// TIA Portal V20 export
FUNCTION_BLOCK "Sequence_1_UnWinder"   // FB118, LAD
TITLE = Sequence
// Sequence template programmend in ladder logic
// stored: IsIECCheckEnabled true, MemoryReserve 100, Namespace Unit1.Em1, SetENOAutomatically true
   VAR
      instSequenceLADControl { ExternalWritable := 'False'} : "LAF_ControlLadSequence";
      instSequenceLADStatus { ExternalWritable := 'False'} : "LAF_StatusLadSequence";
      statPulse { ExternalWritable := 'False'} : Array[0..999] of Bool;
      statTonTimer { ExternalWritable := 'False'} : Array[0..999] of TON_TIME;
   END_VAR
   VAR_TEMP
      tempCustomerAction : Bool;   // Placeholder for possible actions
      tempDo_nothing_and_wait_for_init : Bool;   // Placeholder for doing nothing
      tempSafeStateCondition : Bool;   // Temp Condition for the equipment module to be in a safe state
   END_VAR
   VAR CONSTANT
      STEP_IDLE : DInt := 1;   // Idle Step
      JOB_1_STEP_01 : DInt := 101;
      JOB_1_STEP_11 : DInt := 111;
      JOB_1_STEP_21 : DInt := 121;
      JOB_1_STEP_31 : DInt := 131;
      JOB_1_STEP_41 : DInt := 141;
      JOB_1_STEP_51 : DInt := 151;
      JOB_1_STEP_61 : DInt := 161;
      JOB_1_STEP_71 : DInt := 171;
      JOB_1_STEP_81 : DInt := 181;
      JOB_1_STEP_91 : DInt := 191;
      JOB_2_STEP_01 : DInt := 201;
      JOB_2_STEP_11 : DInt := 211;
      JOB_2_STEP_21 : DInt := 221;
      JOB_2_STEP_31 : DInt := 231;
      JOB_2_STEP_41 : DInt := 241;
      JOB_2_STEP_51 : DInt := 251;
      JOB_2_STEP_61 : DInt := 261;
      JOB_2_STEP_71 : DInt := 271;
      JOB_2_STEP_81 : DInt := 281;
      JOB_2_STEP_91 : DInt := 291;
      JOB_3_STEP_01 : DInt := 301;
      JOB_3_STEP_11 : DInt := 311;
      JOB_3_STEP_21 : DInt := 321;
      JOB_3_STEP_31 : DInt := 331;
      JOB_3_STEP_41 : DInt := 341;
      JOB_3_STEP_51 : DInt := 351;
      JOB_3_STEP_61 : DInt := 361;
      JOB_3_STEP_71 : DInt := 371;
      JOB_3_STEP_81 : DInt := 381;
      JOB_3_STEP_91 : DInt := 391;
      JOB_4_STEP_01 : DInt := 401;
      JOB_4_STEP_11 : DInt := 411;
      JOB_4_STEP_21 : DInt := 421;
      JOB_4_STEP_31 : DInt := 431;
      JOB_4_STEP_41 : DInt := 441;
      JOB_4_STEP_51 : DInt := 451;
      JOB_4_STEP_61 : DInt := 461;
      JOB_4_STEP_71 : DInt := 471;
      JOB_4_STEP_81 : DInt := 481;
      JOB_4_STEP_91 : DInt := 491;
      STEP_IMMEDIATE_STOP : DInt := 901;   // Step executed when an immediate stop command is triggered for the sequence (i.e. when unit is in state aborting)
      SeqDelayTime : Time := T#100ms;
      SeqNoDelayTime : Time;
      SeqReWindingTime : Time := T#3s;
      TRUE : Bool := TRUE;
      FALSE : Bool := FALSE;
   END_VAR
   VAR_TEMP   // added for the SCL form of the ladder/FBD networks
      _w1 : Bool;
   END_VAR
BEGIN

REGION Network 1: BLOCK INFO HEADER
   // (company) / (C) Copyright (year)
   // ---------------------------------------------------------------------------------
   // Title:                             (Title of this block)
   // Comment/Function: (that is implemented in the block)
   // Library/Family:           (that the source is dedicated to)
   // Author:                        (department / person in charge / contact)
   // Target System:          (test system with FW version)
   // Engineering:              TIA Portal (SW version)
   // Restrictions:               (OB types, etc.)
   // Requirements:           (hardware, technological package, etc.)
   // ---------------------------------------------------------------------------------
   // Change log table:
   // Version          | Date             | Signature      | Expert in charge  | Changes applied ------------------------|----------------------|-------------------------|--------------------------------|-----------------------
   // 001.000.000 | yyyy-mm-dd | 0x00000000 | (name of expert) | First released version
END_REGION

REGION Network 2: DESCRIPTION
   // This is a template block provided by the Automation Framework. It can be used to create an own project.
   // The Block Info Header is prepared to put in your own data.
   // Description of the block could be added here and the docu created by Code2Docu.
END_REGION

REGION Network 3: ******************** CONTROL ********************
END_REGION

REGION Network 4: Sequence Control
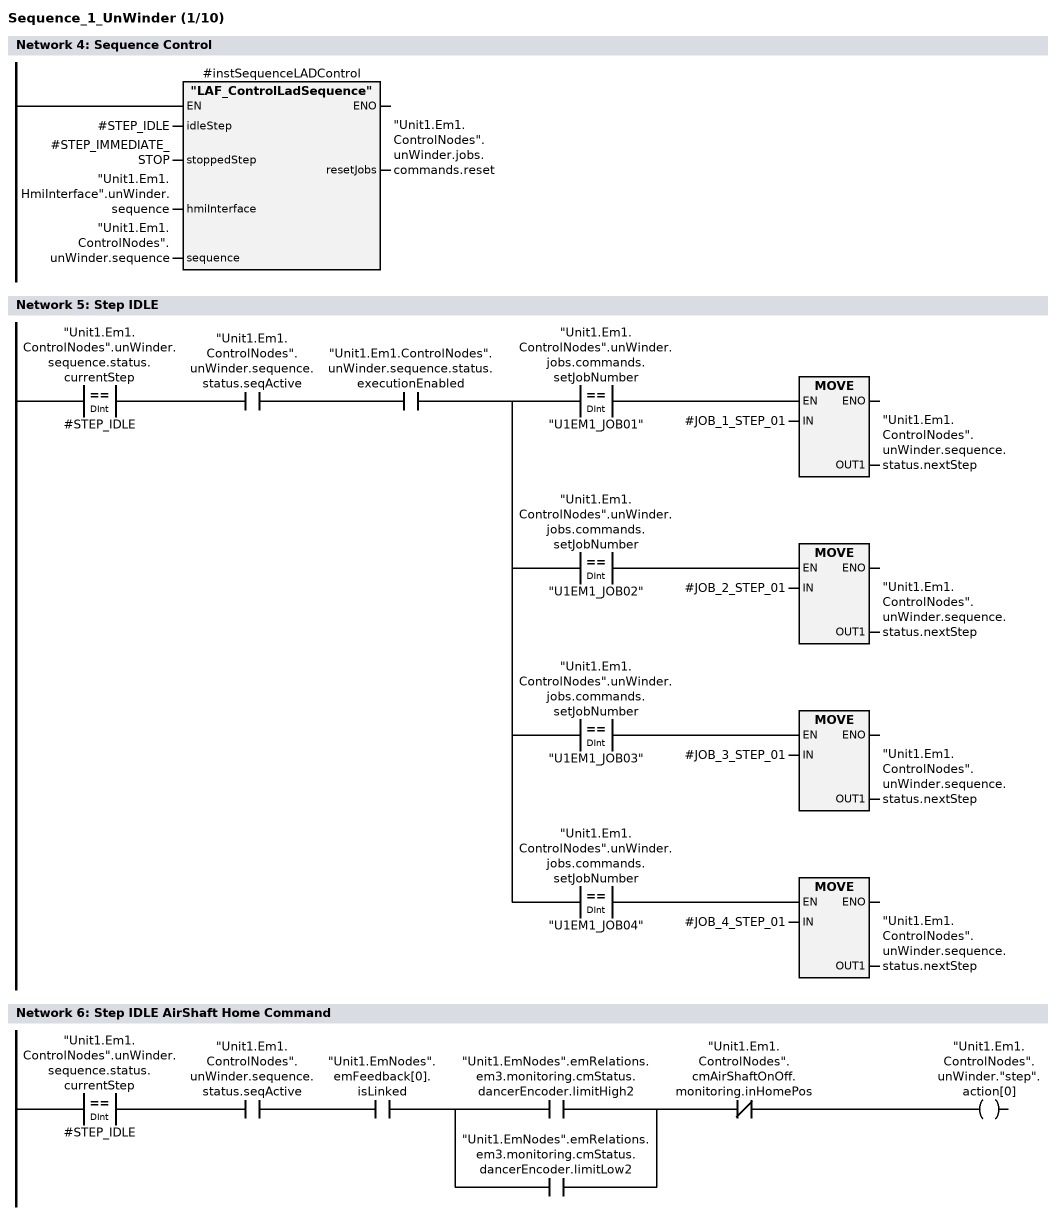
   RUNG wire#powerrail
      #instSequenceLADControl(idleStep := #STEP_IDLE, stoppedStep := #STEP_IMMEDIATE_STOP, hmiInterface := "Unit1.Em1.HmiInterface".unWinder.sequence, sequence := "Unit1.Em1.ControlNodes".unWinder.sequence, resetJobs => "Unit1.Em1.ControlNodes".unWinder.jobs.commands.reset)
   END_RUNG
   // the same network as SCL:
   #instSequenceLADControl(idleStep := #STEP_IDLE,   // "LAF_ControlLadSequence"
                           stoppedStep := #STEP_IMMEDIATE_STOP,
                           hmiInterface := "Unit1.Em1.HmiInterface".unWinder.sequence,
                           sequence := "Unit1.Em1.ControlNodes".unWinder.sequence,
                           resetJobs => "Unit1.Em1.ControlNodes".unWinder.jobs.commands.reset);
END_REGION

REGION Network 5: Step IDLE
   RUNG wire#powerrail
      { S7_Templates := "SrcType := DInt" } EQ_Contact(in1 := "Unit1.Em1.ControlNodes".unWinder.sequence.status.currentStep, in2 := #STEP_IDLE)
      Contact( "Unit1.Em1.ControlNodes".unWinder.sequence.status.seqActive )
      Contact( "Unit1.Em1.ControlNodes".unWinder.sequence.status.executionEnabled )
      wire#w1
      { S7_Templates := "SrcType := DInt" } EQ_Contact(in1 := "Unit1.Em1.ControlNodes".unWinder.jobs.commands.setJobNumber, in2 := "U1EM1_JOB01")
      Move(in := #JOB_1_STEP_01, out1 => "Unit1.Em1.ControlNodes".unWinder.sequence.status.nextStep)
   END_RUNG
   RUNG wire#w1
      { S7_Templates := "SrcType := DInt" } EQ_Contact(in1 := "Unit1.Em1.ControlNodes".unWinder.jobs.commands.setJobNumber, in2 := "U1EM1_JOB02")
      Move(in := #JOB_2_STEP_01, out1 => "Unit1.Em1.ControlNodes".unWinder.sequence.status.nextStep)
   END_RUNG
   RUNG wire#w1
      { S7_Templates := "SrcType := DInt" } EQ_Contact(in1 := "Unit1.Em1.ControlNodes".unWinder.jobs.commands.setJobNumber, in2 := "U1EM1_JOB03")
      Move(in := #JOB_3_STEP_01, out1 => "Unit1.Em1.ControlNodes".unWinder.sequence.status.nextStep)
   END_RUNG
   RUNG wire#w1
      { S7_Templates := "SrcType := DInt" } EQ_Contact(in1 := "Unit1.Em1.ControlNodes".unWinder.jobs.commands.setJobNumber, in2 := "U1EM1_JOB04")
      Move(in := #JOB_4_STEP_01, out1 => "Unit1.Em1.ControlNodes".unWinder.sequence.status.nextStep)
   END_RUNG
   // the same network as SCL:
   #_w1 := ("Unit1.Em1.ControlNodes".unWinder.sequence.status.currentStep = #STEP_IDLE) AND "Unit1.Em1.ControlNodes".unWinder.sequence.status.seqActive AND "Unit1.Em1.ControlNodes".unWinder.sequence.status.executionEnabled;
   IF #_w1 AND ("Unit1.Em1.ControlNodes".unWinder.jobs.commands.setJobNumber = "U1EM1_JOB01") THEN
       "Unit1.Em1.ControlNodes".unWinder.sequence.status.nextStep := #JOB_1_STEP_01;
   END_IF;
   IF #_w1 AND ("Unit1.Em1.ControlNodes".unWinder.jobs.commands.setJobNumber = "U1EM1_JOB02") THEN
       "Unit1.Em1.ControlNodes".unWinder.sequence.status.nextStep := #JOB_2_STEP_01;
   END_IF;
   IF #_w1 AND ("Unit1.Em1.ControlNodes".unWinder.jobs.commands.setJobNumber = "U1EM1_JOB03") THEN
       "Unit1.Em1.ControlNodes".unWinder.sequence.status.nextStep := #JOB_3_STEP_01;
   END_IF;
   IF #_w1 AND ("Unit1.Em1.ControlNodes".unWinder.jobs.commands.setJobNumber = "U1EM1_JOB04") THEN
       "Unit1.Em1.ControlNodes".unWinder.sequence.status.nextStep := #JOB_4_STEP_01;
   END_IF;
END_REGION

REGION Network 6: Step IDLE AirShaft Home Command
   RUNG wire#powerrail
      { S7_Templates := "SrcType := DInt" } EQ_Contact(in1 := "Unit1.Em1.ControlNodes".unWinder.sequence.status.currentStep, in2 := #STEP_IDLE)
      Contact( "Unit1.Em1.ControlNodes".unWinder.sequence.status.seqActive )
      Contact( "Unit1.EmNodes".emFeedback[0].isLinked )
      wire#w1
      Contact( "Unit1.EmNodes".emRelations.em3.monitoring.cmStatus.dancerEncoder.limitHigh2 )
      wire#w2
      I_Contact( "Unit1.Em1.ControlNodes".cmAirShaftOnOff.monitoring.inHomePos )
      Coil( "Unit1.Em1.ControlNodes".unWinder."step".action[0] )
   END_RUNG
   RUNG wire#w1
      Contact( "Unit1.EmNodes".emRelations.em3.monitoring.cmStatus.dancerEncoder.limitLow2 )
   END_RUNG wire#w2
   // the same network as SCL:
   "Unit1.Em1.ControlNodes".unWinder."step".action[0] := ("Unit1.Em1.ControlNodes".unWinder.sequence.status.currentStep = #STEP_IDLE) AND "Unit1.Em1.ControlNodes".unWinder.sequence.status.seqActive AND "Unit1.EmNodes".emFeedback[0].isLinked AND ("Unit1.EmNodes".emRelations.em3.monitoring.cmStatus.dancerEncoder.limitHigh2 OR "Unit1.EmNodes".emRelations.em3.monitoring.cmStatus.dancerEncoder.limitLow2) AND NOT "Unit1.Em1.ControlNodes".cmAirShaftOnOff.monitoring.inHomePos;
END_REGION

REGION Network 7: ******************** JOB[1] EM INITIALIZED ********************
END_REGION

REGION Network 8: Step[101] : JOB[1] Condition
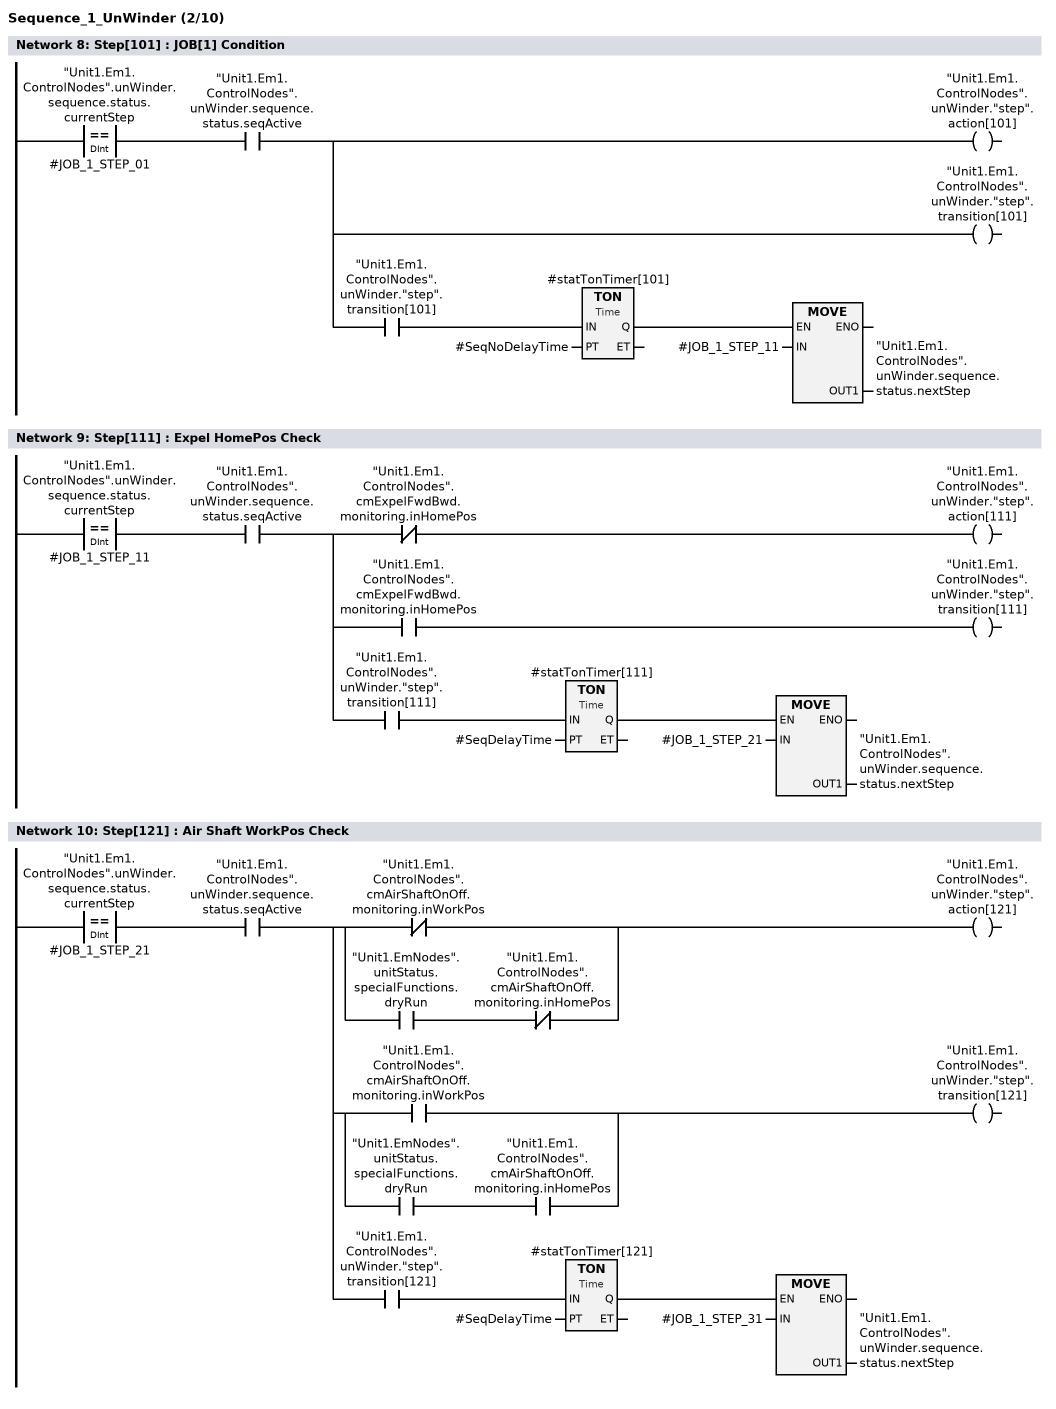
   RUNG wire#powerrail
      { S7_Templates := "SrcType := DInt" } EQ_Contact(in1 := "Unit1.Em1.ControlNodes".unWinder.sequence.status.currentStep, in2 := #JOB_1_STEP_01)
      Contact( "Unit1.Em1.ControlNodes".unWinder.sequence.status.seqActive )
      wire#w1
      Coil( "Unit1.Em1.ControlNodes".unWinder."step".action[101] )
   END_RUNG
   RUNG wire#w1
      Coil( "Unit1.Em1.ControlNodes".unWinder."step".transition[101] )
   END_RUNG
   RUNG wire#w1
      Contact( "Unit1.Em1.ControlNodes".unWinder."step".transition[101] )
      { S7_Templates := "time_type := Time" } #statTonTimer[101].TON(pt := #SeqNoDelayTime, et =>)
      Move(in := #JOB_1_STEP_11, out1 => "Unit1.Em1.ControlNodes".unWinder.sequence.status.nextStep)
   END_RUNG
   // the same network as SCL:
   "Unit1.Em1.ControlNodes".unWinder."step".action[101] := ("Unit1.Em1.ControlNodes".unWinder.sequence.status.currentStep = #JOB_1_STEP_01) AND "Unit1.Em1.ControlNodes".unWinder.sequence.status.seqActive;
   "Unit1.Em1.ControlNodes".unWinder."step".transition[101] := ("Unit1.Em1.ControlNodes".unWinder.sequence.status.currentStep = #JOB_1_STEP_01) AND "Unit1.Em1.ControlNodes".unWinder.sequence.status.seqActive;
   #statTonTimer[101].TON(IN := ("Unit1.Em1.ControlNodes".unWinder.sequence.status.currentStep = #JOB_1_STEP_01) AND "Unit1.Em1.ControlNodes".unWinder.sequence.status.seqActive AND "Unit1.Em1.ControlNodes".unWinder."step".transition[101],
                          PT := #SeqNoDelayTime);
   IF #statTonTimer[101].Q THEN
       "Unit1.Em1.ControlNodes".unWinder.sequence.status.nextStep := #JOB_1_STEP_11;
   END_IF;
END_REGION

REGION Network 9: Step[111] : Expel HomePos Check
   RUNG wire#powerrail
      { S7_Templates := "SrcType := DInt" } EQ_Contact(in1 := "Unit1.Em1.ControlNodes".unWinder.sequence.status.currentStep, in2 := #JOB_1_STEP_11)
      Contact( "Unit1.Em1.ControlNodes".unWinder.sequence.status.seqActive )
      wire#w1
      I_Contact( "Unit1.Em1.ControlNodes".cmExpelFwdBwd.monitoring.inHomePos )
      Coil( "Unit1.Em1.ControlNodes".unWinder."step".action[111] )
   END_RUNG
   RUNG wire#w1
      Contact( "Unit1.Em1.ControlNodes".cmExpelFwdBwd.monitoring.inHomePos )
      Coil( "Unit1.Em1.ControlNodes".unWinder."step".transition[111] )
   END_RUNG
   RUNG wire#w1
      Contact( "Unit1.Em1.ControlNodes".unWinder."step".transition[111] )
      { S7_Templates := "time_type := Time" } #statTonTimer[111].TON(pt := #SeqDelayTime, et =>)
      Move(in := #JOB_1_STEP_21, out1 => "Unit1.Em1.ControlNodes".unWinder.sequence.status.nextStep)
   END_RUNG
   // the same network as SCL:
   #_w1 := ("Unit1.Em1.ControlNodes".unWinder.sequence.status.currentStep = #JOB_1_STEP_11) AND "Unit1.Em1.ControlNodes".unWinder.sequence.status.seqActive;
   "Unit1.Em1.ControlNodes".unWinder."step".action[111] := #_w1 AND NOT "Unit1.Em1.ControlNodes".cmExpelFwdBwd.monitoring.inHomePos;
   "Unit1.Em1.ControlNodes".unWinder."step".transition[111] := #_w1 AND "Unit1.Em1.ControlNodes".cmExpelFwdBwd.monitoring.inHomePos;
   #statTonTimer[111].TON(IN := #_w1 AND "Unit1.Em1.ControlNodes".unWinder."step".transition[111],
                          PT := #SeqDelayTime);
   IF #statTonTimer[111].Q THEN
       "Unit1.Em1.ControlNodes".unWinder.sequence.status.nextStep := #JOB_1_STEP_21;
   END_IF;
END_REGION

REGION Network 10: Step[121] : Air Shaft WorkPos Check
   RUNG wire#powerrail
      { S7_Templates := "SrcType := DInt" } EQ_Contact(in1 := "Unit1.Em1.ControlNodes".unWinder.sequence.status.currentStep, in2 := #JOB_1_STEP_21)
      Contact( "Unit1.Em1.ControlNodes".unWinder.sequence.status.seqActive )
      wire#w1
      I_Contact( "Unit1.Em1.ControlNodes".cmAirShaftOnOff.monitoring.inWorkPos )
      wire#w2
      Coil( "Unit1.Em1.ControlNodes".unWinder."step".action[121] )
   END_RUNG
   RUNG wire#w1
      Contact( "Unit1.EmNodes".unitStatus.specialFunctions.dryRun )
      I_Contact( "Unit1.Em1.ControlNodes".cmAirShaftOnOff.monitoring.inHomePos )
   END_RUNG wire#w2
   RUNG wire#w1
      Contact( "Unit1.Em1.ControlNodes".cmAirShaftOnOff.monitoring.inWorkPos )
      wire#w3
      Coil( "Unit1.Em1.ControlNodes".unWinder."step".transition[121] )
   END_RUNG
   RUNG wire#w1
      Contact( "Unit1.EmNodes".unitStatus.specialFunctions.dryRun )
      Contact( "Unit1.Em1.ControlNodes".cmAirShaftOnOff.monitoring.inHomePos )
   END_RUNG wire#w3
   RUNG wire#w1
      Contact( "Unit1.Em1.ControlNodes".unWinder."step".transition[121] )
      { S7_Templates := "time_type := Time" } #statTonTimer[121].TON(pt := #SeqDelayTime, et =>)
      Move(in := #JOB_1_STEP_31, out1 => "Unit1.Em1.ControlNodes".unWinder.sequence.status.nextStep)
   END_RUNG
   // the same network as SCL:
   #_w1 := ("Unit1.Em1.ControlNodes".unWinder.sequence.status.currentStep = #JOB_1_STEP_21) AND "Unit1.Em1.ControlNodes".unWinder.sequence.status.seqActive;
   "Unit1.Em1.ControlNodes".unWinder."step".action[121] := #_w1 AND (NOT "Unit1.Em1.ControlNodes".cmAirShaftOnOff.monitoring.inWorkPos OR ("Unit1.EmNodes".unitStatus.specialFunctions.dryRun AND NOT "Unit1.Em1.ControlNodes".cmAirShaftOnOff.monitoring.inHomePos));
   "Unit1.Em1.ControlNodes".unWinder."step".transition[121] := #_w1 AND ("Unit1.Em1.ControlNodes".cmAirShaftOnOff.monitoring.inWorkPos OR ("Unit1.EmNodes".unitStatus.specialFunctions.dryRun AND "Unit1.Em1.ControlNodes".cmAirShaftOnOff.monitoring.inHomePos));
   #statTonTimer[121].TON(IN := #_w1 AND "Unit1.Em1.ControlNodes".unWinder."step".transition[121],
                          PT := #SeqDelayTime);
   IF #statTonTimer[121].Q THEN
       "Unit1.Em1.ControlNodes".unWinder.sequence.status.nextStep := #JOB_1_STEP_31;
   END_IF;
END_REGION

REGION Network 11: Step[131] : Radius Measure Check
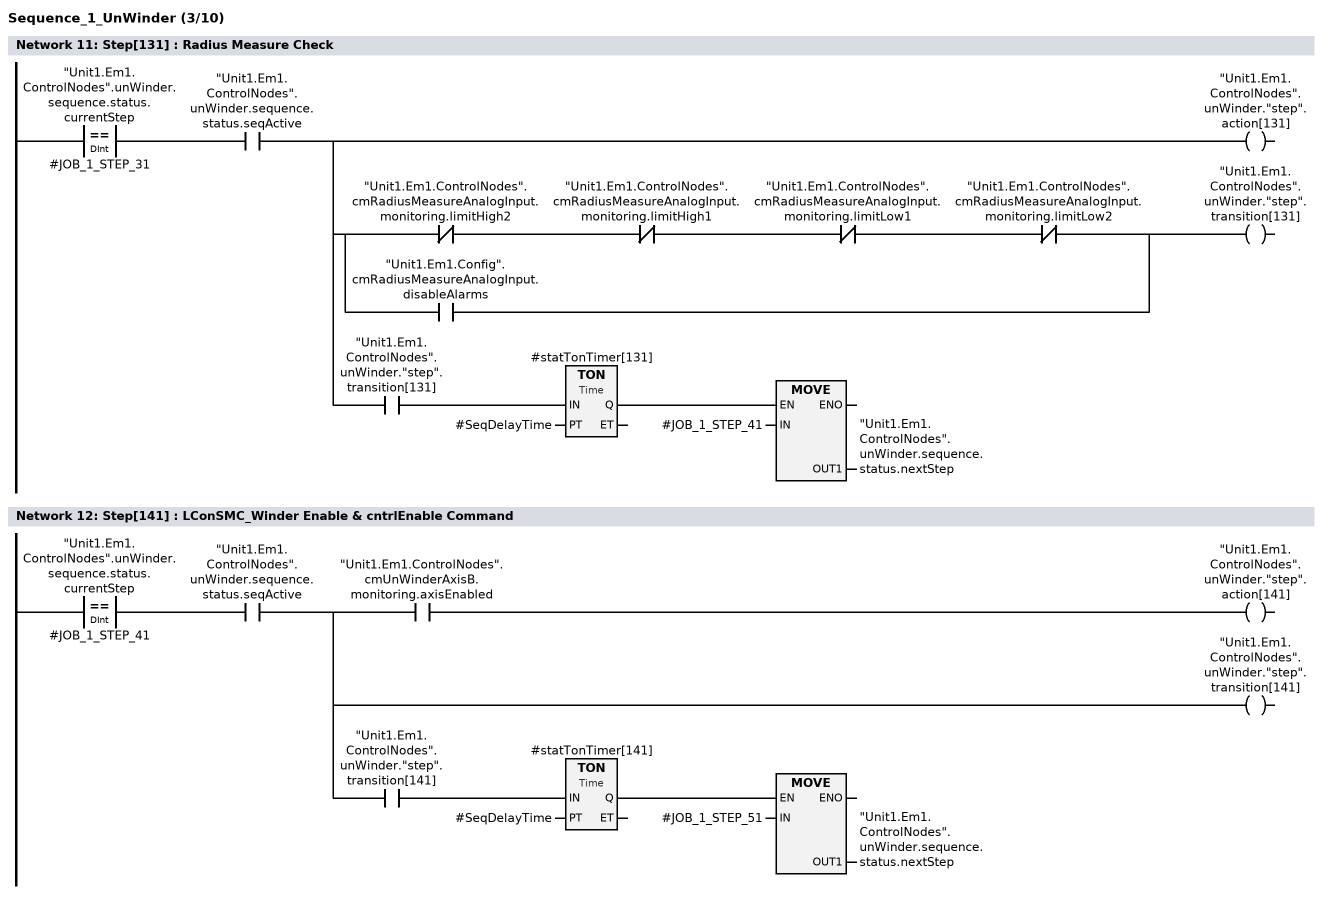
   RUNG wire#powerrail
      { S7_Templates := "SrcType := DInt" } EQ_Contact(in1 := "Unit1.Em1.ControlNodes".unWinder.sequence.status.currentStep, in2 := #JOB_1_STEP_31)
      Contact( "Unit1.Em1.ControlNodes".unWinder.sequence.status.seqActive )
      wire#w1
      Coil( "Unit1.Em1.ControlNodes".unWinder."step".action[131] )
   END_RUNG
   RUNG wire#w1
      I_Contact( "Unit1.Em1.ControlNodes".cmRadiusMeasureAnalogInput.monitoring.limitHigh2 )
      I_Contact( "Unit1.Em1.ControlNodes".cmRadiusMeasureAnalogInput.monitoring.limitHigh1 )
      I_Contact( "Unit1.Em1.ControlNodes".cmRadiusMeasureAnalogInput.monitoring.limitLow1 )
      I_Contact( "Unit1.Em1.ControlNodes".cmRadiusMeasureAnalogInput.monitoring.limitLow2 )
      wire#w2
      Coil( "Unit1.Em1.ControlNodes".unWinder."step".transition[131] )
   END_RUNG
   RUNG wire#w1
      Contact( "Unit1.Em1.Config".cmRadiusMeasureAnalogInput.disableAlarms )
   END_RUNG wire#w2
   RUNG wire#w1
      Contact( "Unit1.Em1.ControlNodes".unWinder."step".transition[131] )
      { S7_Templates := "time_type := Time" } #statTonTimer[131].TON(pt := #SeqDelayTime, et =>)
      Move(in := #JOB_1_STEP_41, out1 => "Unit1.Em1.ControlNodes".unWinder.sequence.status.nextStep)
   END_RUNG
   // the same network as SCL:
   "Unit1.Em1.ControlNodes".unWinder."step".action[131] := ("Unit1.Em1.ControlNodes".unWinder.sequence.status.currentStep = #JOB_1_STEP_31) AND "Unit1.Em1.ControlNodes".unWinder.sequence.status.seqActive;
   "Unit1.Em1.ControlNodes".unWinder."step".transition[131] := ("Unit1.Em1.ControlNodes".unWinder.sequence.status.currentStep = #JOB_1_STEP_31) AND "Unit1.Em1.ControlNodes".unWinder.sequence.status.seqActive AND ((NOT "Unit1.Em1.ControlNodes".cmRadiusMeasureAnalogInput.monitoring.limitHigh2 AND NOT "Unit1.Em1.ControlNodes".cmRadiusMeasureAnalogInput.monitoring.limitHigh1 AND NOT "Unit1.Em1.ControlNodes".cmRadiusMeasureAnalogInput.monitoring.limitLow1 AND NOT "Unit1.Em1.ControlNodes".cmRadiusMeasureAnalogInput.monitoring.limitLow2) OR "Unit1.Em1.Config".cmRadiusMeasureAnalogInput.disableAlarms);
   #statTonTimer[131].TON(IN := ("Unit1.Em1.ControlNodes".unWinder.sequence.status.currentStep = #JOB_1_STEP_31) AND "Unit1.Em1.ControlNodes".unWinder.sequence.status.seqActive AND "Unit1.Em1.ControlNodes".unWinder."step".transition[131],
                          PT := #SeqDelayTime);
   IF #statTonTimer[131].Q THEN
       "Unit1.Em1.ControlNodes".unWinder.sequence.status.nextStep := #JOB_1_STEP_41;
   END_IF;
END_REGION

REGION Network 12: Step[141] : LConSMC_Winder Enable & cntrlEnable Command
   RUNG wire#powerrail
      { S7_Templates := "SrcType := DInt" } EQ_Contact(in1 := "Unit1.Em1.ControlNodes".unWinder.sequence.status.currentStep, in2 := #JOB_1_STEP_41)
      Contact( "Unit1.Em1.ControlNodes".unWinder.sequence.status.seqActive )
      wire#w1
      Contact( "Unit1.Em1.ControlNodes".cmUnWinderAxisB.monitoring.axisEnabled )
      Coil( "Unit1.Em1.ControlNodes".unWinder."step".action[141] )
   END_RUNG
   RUNG wire#w1
      Coil( "Unit1.Em1.ControlNodes".unWinder."step".transition[141] )
   END_RUNG
   RUNG wire#w1
      Contact( "Unit1.Em1.ControlNodes".unWinder."step".transition[141] )
      { S7_Templates := "time_type := Time" } #statTonTimer[141].TON(pt := #SeqDelayTime, et =>)
      Move(in := #JOB_1_STEP_51, out1 => "Unit1.Em1.ControlNodes".unWinder.sequence.status.nextStep)
   END_RUNG
   // the same network as SCL:
   #_w1 := ("Unit1.Em1.ControlNodes".unWinder.sequence.status.currentStep = #JOB_1_STEP_41) AND "Unit1.Em1.ControlNodes".unWinder.sequence.status.seqActive;
   "Unit1.Em1.ControlNodes".unWinder."step".action[141] := #_w1 AND "Unit1.Em1.ControlNodes".cmUnWinderAxisB.monitoring.axisEnabled;
   "Unit1.Em1.ControlNodes".unWinder."step".transition[141] := #_w1;
   #statTonTimer[141].TON(IN := #_w1 AND "Unit1.Em1.ControlNodes".unWinder."step".transition[141],
                          PT := #SeqDelayTime);
   IF #statTonTimer[141].Q THEN
       "Unit1.Em1.ControlNodes".unWinder.sequence.status.nextStep := #JOB_1_STEP_51;
   END_IF;
END_REGION

REGION Network 13: Step[151] : Web Guide EPC Mode Check
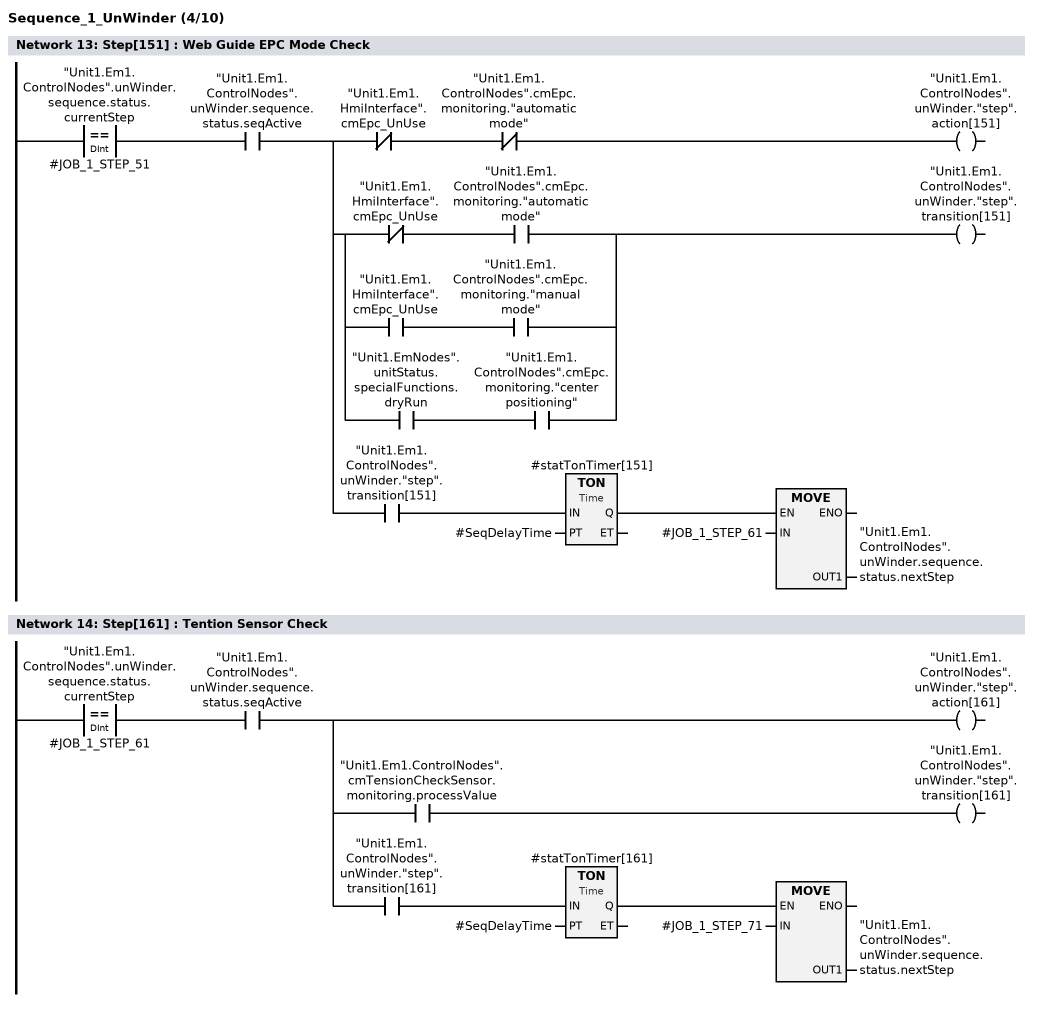
   RUNG wire#powerrail
      { S7_Templates := "SrcType := DInt" } EQ_Contact(in1 := "Unit1.Em1.ControlNodes".unWinder.sequence.status.currentStep, in2 := #JOB_1_STEP_51)
      Contact( "Unit1.Em1.ControlNodes".unWinder.sequence.status.seqActive )
      wire#w1
      I_Contact( "Unit1.Em1.HmiInterface".cmEpc_UnUse )
      I_Contact( "Unit1.Em1.ControlNodes".cmEpc.monitoring."automatic mode" )
      Coil( "Unit1.Em1.ControlNodes".unWinder."step".action[151] )
   END_RUNG
   RUNG wire#w1
      I_Contact( "Unit1.Em1.HmiInterface".cmEpc_UnUse )
      Contact( "Unit1.Em1.ControlNodes".cmEpc.monitoring."automatic mode" )
      wire#w2
      Coil( "Unit1.Em1.ControlNodes".unWinder."step".transition[151] )
   END_RUNG
   RUNG wire#w1
      Contact( "Unit1.Em1.HmiInterface".cmEpc_UnUse )
      Contact( "Unit1.Em1.ControlNodes".cmEpc.monitoring."manual mode" )
   END_RUNG wire#w2
   RUNG wire#w1
      Contact( "Unit1.EmNodes".unitStatus.specialFunctions.dryRun )
      Contact( "Unit1.Em1.ControlNodes".cmEpc.monitoring."center positioning" )
   END_RUNG wire#w2
   RUNG wire#w1
      Contact( "Unit1.Em1.ControlNodes".unWinder."step".transition[151] )
      { S7_Templates := "time_type := Time" } #statTonTimer[151].TON(pt := #SeqDelayTime, et =>)
      Move(in := #JOB_1_STEP_61, out1 => "Unit1.Em1.ControlNodes".unWinder.sequence.status.nextStep)
   END_RUNG
   // the same network as SCL:
   #_w1 := ("Unit1.Em1.ControlNodes".unWinder.sequence.status.currentStep = #JOB_1_STEP_51) AND "Unit1.Em1.ControlNodes".unWinder.sequence.status.seqActive;
   "Unit1.Em1.ControlNodes".unWinder."step".action[151] := #_w1 AND NOT "Unit1.Em1.HmiInterface".cmEpc_UnUse AND NOT "Unit1.Em1.ControlNodes".cmEpc.monitoring."automatic mode";
   "Unit1.Em1.ControlNodes".unWinder."step".transition[151] := #_w1 AND ((NOT "Unit1.Em1.HmiInterface".cmEpc_UnUse AND "Unit1.Em1.ControlNodes".cmEpc.monitoring."automatic mode") OR ("Unit1.Em1.HmiInterface".cmEpc_UnUse AND "Unit1.Em1.ControlNodes".cmEpc.monitoring."manual mode") OR ("Unit1.EmNodes".unitStatus.specialFunctions.dryRun AND "Unit1.Em1.ControlNodes".cmEpc.monitoring."center positioning"));
   #statTonTimer[151].TON(IN := #_w1 AND "Unit1.Em1.ControlNodes".unWinder."step".transition[151],
                          PT := #SeqDelayTime);
   IF #statTonTimer[151].Q THEN
       "Unit1.Em1.ControlNodes".unWinder.sequence.status.nextStep := #JOB_1_STEP_61;
   END_IF;
END_REGION

REGION Network 14: Step[161] : Tention Sensor Check
   RUNG wire#powerrail
      { S7_Templates := "SrcType := DInt" } EQ_Contact(in1 := "Unit1.Em1.ControlNodes".unWinder.sequence.status.currentStep, in2 := #JOB_1_STEP_61)
      Contact( "Unit1.Em1.ControlNodes".unWinder.sequence.status.seqActive )
      wire#w1
      Coil( "Unit1.Em1.ControlNodes".unWinder."step".action[161] )
   END_RUNG
   RUNG wire#w1
      Contact( "Unit1.Em1.ControlNodes".cmTensionCheckSensor.monitoring.processValue )
      Coil( "Unit1.Em1.ControlNodes".unWinder."step".transition[161] )
   END_RUNG
   RUNG wire#w1
      Contact( "Unit1.Em1.ControlNodes".unWinder."step".transition[161] )
      { S7_Templates := "time_type := Time" } #statTonTimer[161].TON(pt := #SeqDelayTime, et =>)
      Move(in := #JOB_1_STEP_71, out1 => "Unit1.Em1.ControlNodes".unWinder.sequence.status.nextStep)
   END_RUNG
   // the same network as SCL:
   "Unit1.Em1.ControlNodes".unWinder."step".action[161] := ("Unit1.Em1.ControlNodes".unWinder.sequence.status.currentStep = #JOB_1_STEP_61) AND "Unit1.Em1.ControlNodes".unWinder.sequence.status.seqActive;
   "Unit1.Em1.ControlNodes".unWinder."step".transition[161] := ("Unit1.Em1.ControlNodes".unWinder.sequence.status.currentStep = #JOB_1_STEP_61) AND "Unit1.Em1.ControlNodes".unWinder.sequence.status.seqActive AND "Unit1.Em1.ControlNodes".cmTensionCheckSensor.monitoring.processValue;
   #statTonTimer[161].TON(IN := ("Unit1.Em1.ControlNodes".unWinder.sequence.status.currentStep = #JOB_1_STEP_61) AND "Unit1.Em1.ControlNodes".unWinder.sequence.status.seqActive AND "Unit1.Em1.ControlNodes".unWinder."step".transition[161],
                          PT := #SeqDelayTime);
   IF #statTonTimer[161].Q THEN
       "Unit1.Em1.ControlNodes".unWinder.sequence.status.nextStep := #JOB_1_STEP_71;
   END_IF;
END_REGION

REGION Network 15: Step[161] : Bobin ID Check
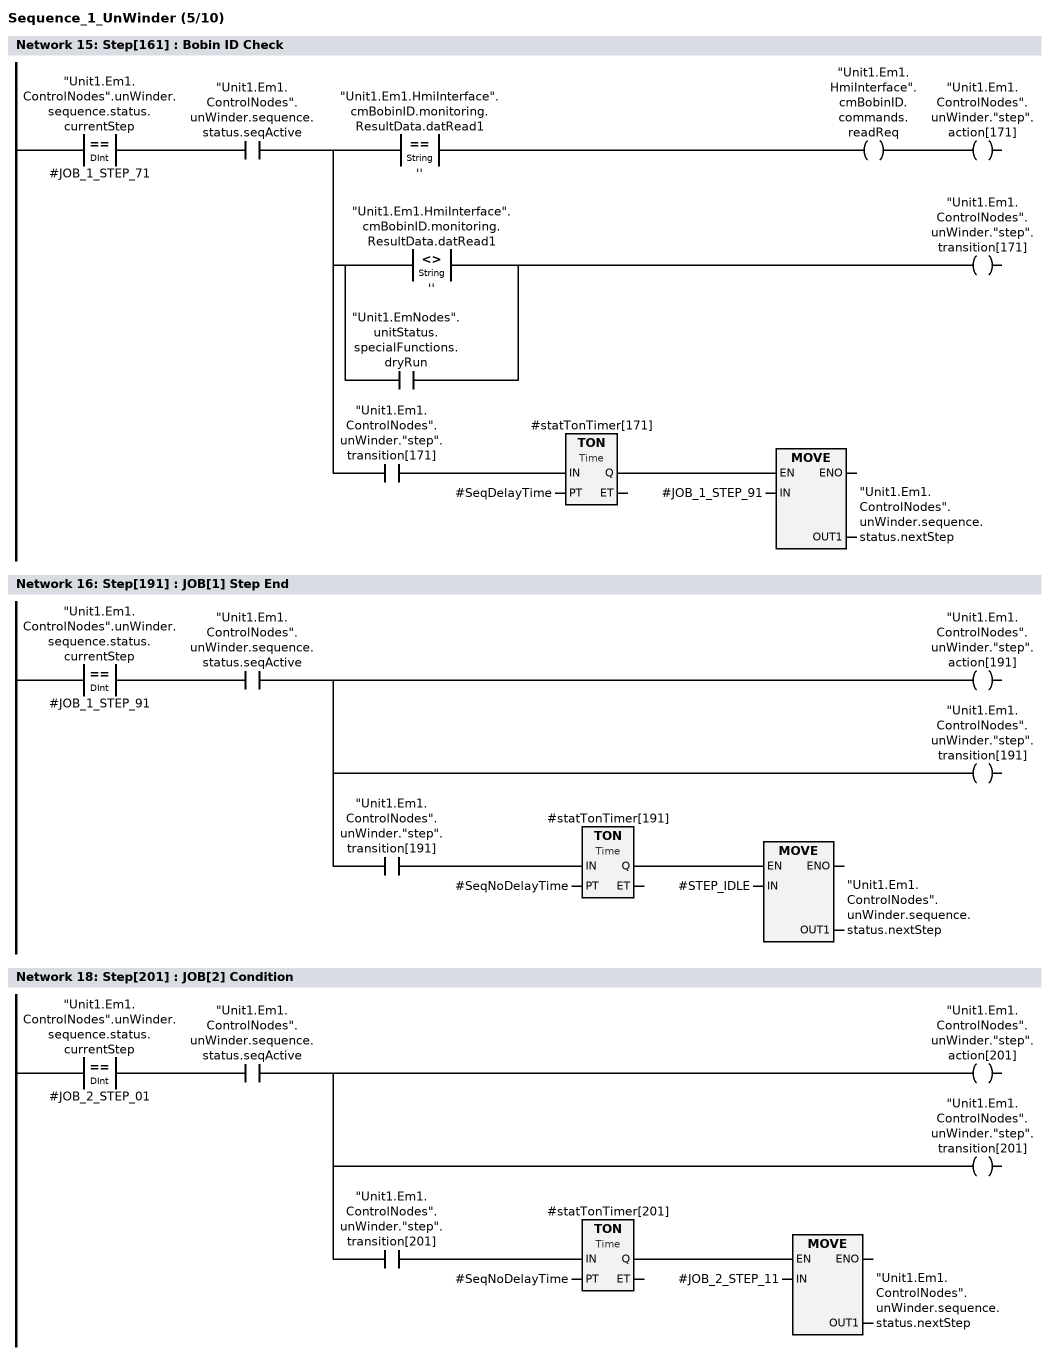
   RUNG wire#powerrail
      { S7_Templates := "SrcType := DInt" } EQ_Contact(in1 := "Unit1.Em1.ControlNodes".unWinder.sequence.status.currentStep, in2 := #JOB_1_STEP_71)
      Contact( "Unit1.Em1.ControlNodes".unWinder.sequence.status.seqActive )
      wire#w1
      { S7_Templates := "SrcType := String" } EQ_Contact(in1 := "Unit1.Em1.HmiInterface".cmBobinID.monitoring.ResultData.datRead1, in2 := '')
      Coil( "Unit1.Em1.HmiInterface".cmBobinID.commands.readReq )
      Coil( "Unit1.Em1.ControlNodes".unWinder."step".action[171] )
   END_RUNG
   RUNG wire#w1
      { S7_Templates := "SrcType := String" } NE_Contact(in1 := "Unit1.Em1.HmiInterface".cmBobinID.monitoring.ResultData.datRead1, in2 := '')
      wire#w2
      Coil( "Unit1.Em1.ControlNodes".unWinder."step".transition[171] )
   END_RUNG
   RUNG wire#w1
      Contact( "Unit1.EmNodes".unitStatus.specialFunctions.dryRun )
   END_RUNG wire#w2
   RUNG wire#w1
      Contact( "Unit1.Em1.ControlNodes".unWinder."step".transition[171] )
      { S7_Templates := "time_type := Time" } #statTonTimer[171].TON(pt := #SeqDelayTime, et =>)
      Move(in := #JOB_1_STEP_91, out1 => "Unit1.Em1.ControlNodes".unWinder.sequence.status.nextStep)
   END_RUNG
   // the same network as SCL:
   #_w1 := ("Unit1.Em1.ControlNodes".unWinder.sequence.status.currentStep = #JOB_1_STEP_71) AND "Unit1.Em1.ControlNodes".unWinder.sequence.status.seqActive;
   "Unit1.Em1.HmiInterface".cmBobinID.commands.readReq := #_w1 AND ("Unit1.Em1.HmiInterface".cmBobinID.monitoring.ResultData.datRead1 = '');
   "Unit1.Em1.ControlNodes".unWinder."step".action[171] := "Unit1.Em1.HmiInterface".cmBobinID.commands.readReq;
   "Unit1.Em1.ControlNodes".unWinder."step".transition[171] := #_w1 AND (("Unit1.Em1.HmiInterface".cmBobinID.monitoring.ResultData.datRead1 <> '') OR "Unit1.EmNodes".unitStatus.specialFunctions.dryRun);
   #statTonTimer[171].TON(IN := #_w1 AND "Unit1.Em1.ControlNodes".unWinder."step".transition[171],
                          PT := #SeqDelayTime);
   IF #statTonTimer[171].Q THEN
       "Unit1.Em1.ControlNodes".unWinder.sequence.status.nextStep := #JOB_1_STEP_91;
   END_IF;
END_REGION

REGION Network 16: Step[191] : JOB[1] Step End
   RUNG wire#powerrail
      { S7_Templates := "SrcType := DInt" } EQ_Contact(in1 := "Unit1.Em1.ControlNodes".unWinder.sequence.status.currentStep, in2 := #JOB_1_STEP_91)
      Contact( "Unit1.Em1.ControlNodes".unWinder.sequence.status.seqActive )
      wire#w1
      Coil( "Unit1.Em1.ControlNodes".unWinder."step".action[191] )
   END_RUNG
   RUNG wire#w1
      Coil( "Unit1.Em1.ControlNodes".unWinder."step".transition[191] )
   END_RUNG
   RUNG wire#w1
      Contact( "Unit1.Em1.ControlNodes".unWinder."step".transition[191] )
      { S7_Templates := "time_type := Time" } #statTonTimer[191].TON(pt := #SeqNoDelayTime, et =>)
      Move(in := #STEP_IDLE, out1 => "Unit1.Em1.ControlNodes".unWinder.sequence.status.nextStep)
   END_RUNG
   // the same network as SCL:
   "Unit1.Em1.ControlNodes".unWinder."step".action[191] := ("Unit1.Em1.ControlNodes".unWinder.sequence.status.currentStep = #JOB_1_STEP_91) AND "Unit1.Em1.ControlNodes".unWinder.sequence.status.seqActive;
   "Unit1.Em1.ControlNodes".unWinder."step".transition[191] := ("Unit1.Em1.ControlNodes".unWinder.sequence.status.currentStep = #JOB_1_STEP_91) AND "Unit1.Em1.ControlNodes".unWinder.sequence.status.seqActive;
   #statTonTimer[191].TON(IN := ("Unit1.Em1.ControlNodes".unWinder.sequence.status.currentStep = #JOB_1_STEP_91) AND "Unit1.Em1.ControlNodes".unWinder.sequence.status.seqActive AND "Unit1.Em1.ControlNodes".unWinder."step".transition[191],
                          PT := #SeqNoDelayTime);
   IF #statTonTimer[191].Q THEN
       "Unit1.Em1.ControlNodes".unWinder.sequence.status.nextStep := #STEP_IDLE;
   END_IF;
END_REGION

REGION Network 17: ******************** JOB[2] UNWINDER RUN ********************
END_REGION

REGION Network 18: Step[201] : JOB[2] Condition
   RUNG wire#powerrail
      { S7_Templates := "SrcType := DInt" } EQ_Contact(in1 := "Unit1.Em1.ControlNodes".unWinder.sequence.status.currentStep, in2 := #JOB_2_STEP_01)
      Contact( "Unit1.Em1.ControlNodes".unWinder.sequence.status.seqActive )
      wire#w1
      Coil( "Unit1.Em1.ControlNodes".unWinder."step".action[201] )
   END_RUNG
   RUNG wire#w1
      Coil( "Unit1.Em1.ControlNodes".unWinder."step".transition[201] )
   END_RUNG
   RUNG wire#w1
      Contact( "Unit1.Em1.ControlNodes".unWinder."step".transition[201] )
      { S7_Templates := "time_type := Time" } #statTonTimer[201].TON(pt := #SeqNoDelayTime, et =>)
      Move(in := #JOB_2_STEP_11, out1 => "Unit1.Em1.ControlNodes".unWinder.sequence.status.nextStep)
   END_RUNG
   // the same network as SCL:
   "Unit1.Em1.ControlNodes".unWinder."step".action[201] := ("Unit1.Em1.ControlNodes".unWinder.sequence.status.currentStep = #JOB_2_STEP_01) AND "Unit1.Em1.ControlNodes".unWinder.sequence.status.seqActive;
   "Unit1.Em1.ControlNodes".unWinder."step".transition[201] := ("Unit1.Em1.ControlNodes".unWinder.sequence.status.currentStep = #JOB_2_STEP_01) AND "Unit1.Em1.ControlNodes".unWinder.sequence.status.seqActive;
   #statTonTimer[201].TON(IN := ("Unit1.Em1.ControlNodes".unWinder.sequence.status.currentStep = #JOB_2_STEP_01) AND "Unit1.Em1.ControlNodes".unWinder.sequence.status.seqActive AND "Unit1.Em1.ControlNodes".unWinder."step".transition[201],
                          PT := #SeqNoDelayTime);
   IF #statTonTimer[201].Q THEN
       "Unit1.Em1.ControlNodes".unWinder.sequence.status.nextStep := #JOB_2_STEP_11;
   END_IF;
END_REGION

REGION Network 19: Step[211] : LConSMC_Winder speedMatch Command
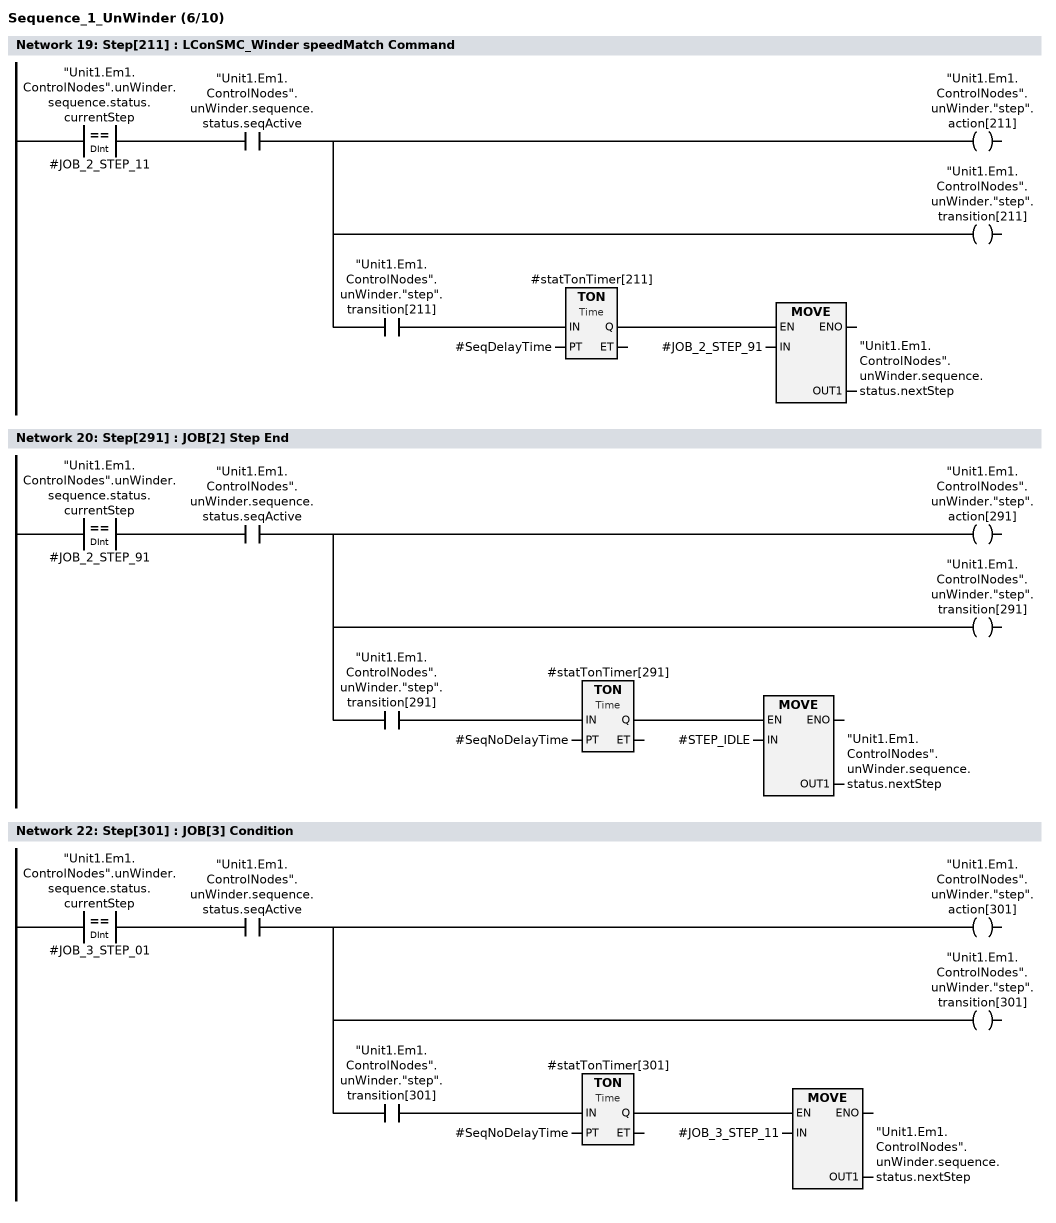
   RUNG wire#powerrail
      { S7_Templates := "SrcType := DInt" } EQ_Contact(in1 := "Unit1.Em1.ControlNodes".unWinder.sequence.status.currentStep, in2 := #JOB_2_STEP_11)
      Contact( "Unit1.Em1.ControlNodes".unWinder.sequence.status.seqActive )
      wire#w1
      Coil( "Unit1.Em1.ControlNodes".unWinder."step".action[211] )
   END_RUNG
   RUNG wire#w1
      Coil( "Unit1.Em1.ControlNodes".unWinder."step".transition[211] )
   END_RUNG
   RUNG wire#w1
      Contact( "Unit1.Em1.ControlNodes".unWinder."step".transition[211] )
      { S7_Templates := "time_type := Time" } #statTonTimer[211].TON(pt := #SeqDelayTime, et =>)
      Move(in := #JOB_2_STEP_91, out1 => "Unit1.Em1.ControlNodes".unWinder.sequence.status.nextStep)
   END_RUNG
   // the same network as SCL:
   "Unit1.Em1.ControlNodes".unWinder."step".action[211] := ("Unit1.Em1.ControlNodes".unWinder.sequence.status.currentStep = #JOB_2_STEP_11) AND "Unit1.Em1.ControlNodes".unWinder.sequence.status.seqActive;
   "Unit1.Em1.ControlNodes".unWinder."step".transition[211] := ("Unit1.Em1.ControlNodes".unWinder.sequence.status.currentStep = #JOB_2_STEP_11) AND "Unit1.Em1.ControlNodes".unWinder.sequence.status.seqActive;
   #statTonTimer[211].TON(IN := ("Unit1.Em1.ControlNodes".unWinder.sequence.status.currentStep = #JOB_2_STEP_11) AND "Unit1.Em1.ControlNodes".unWinder.sequence.status.seqActive AND "Unit1.Em1.ControlNodes".unWinder."step".transition[211],
                          PT := #SeqDelayTime);
   IF #statTonTimer[211].Q THEN
       "Unit1.Em1.ControlNodes".unWinder.sequence.status.nextStep := #JOB_2_STEP_91;
   END_IF;
END_REGION

REGION Network 20: Step[291] : JOB[2] Step End
   RUNG wire#powerrail
      { S7_Templates := "SrcType := DInt" } EQ_Contact(in1 := "Unit1.Em1.ControlNodes".unWinder.sequence.status.currentStep, in2 := #JOB_2_STEP_91)
      Contact( "Unit1.Em1.ControlNodes".unWinder.sequence.status.seqActive )
      wire#w1
      Coil( "Unit1.Em1.ControlNodes".unWinder."step".action[291] )
   END_RUNG
   RUNG wire#w1
      Coil( "Unit1.Em1.ControlNodes".unWinder."step".transition[291] )
   END_RUNG
   RUNG wire#w1
      Contact( "Unit1.Em1.ControlNodes".unWinder."step".transition[291] )
      { S7_Templates := "time_type := Time" } #statTonTimer[291].TON(pt := #SeqNoDelayTime, et =>)
      Move(in := #STEP_IDLE, out1 => "Unit1.Em1.ControlNodes".unWinder.sequence.status.nextStep)
   END_RUNG
   // the same network as SCL:
   "Unit1.Em1.ControlNodes".unWinder."step".action[291] := ("Unit1.Em1.ControlNodes".unWinder.sequence.status.currentStep = #JOB_2_STEP_91) AND "Unit1.Em1.ControlNodes".unWinder.sequence.status.seqActive;
   "Unit1.Em1.ControlNodes".unWinder."step".transition[291] := ("Unit1.Em1.ControlNodes".unWinder.sequence.status.currentStep = #JOB_2_STEP_91) AND "Unit1.Em1.ControlNodes".unWinder.sequence.status.seqActive;
   #statTonTimer[291].TON(IN := ("Unit1.Em1.ControlNodes".unWinder.sequence.status.currentStep = #JOB_2_STEP_91) AND "Unit1.Em1.ControlNodes".unWinder.sequence.status.seqActive AND "Unit1.Em1.ControlNodes".unWinder."step".transition[291],
                          PT := #SeqNoDelayTime);
   IF #statTonTimer[291].Q THEN
       "Unit1.Em1.ControlNodes".unWinder.sequence.status.nextStep := #STEP_IDLE;
   END_IF;
END_REGION

REGION Network 21: ******************** JOB[3] UNWINDER STOP ********************
END_REGION

REGION Network 22: Step[301] : JOB[3] Condition
   RUNG wire#powerrail
      { S7_Templates := "SrcType := DInt" } EQ_Contact(in1 := "Unit1.Em1.ControlNodes".unWinder.sequence.status.currentStep, in2 := #JOB_3_STEP_01)
      Contact( "Unit1.Em1.ControlNodes".unWinder.sequence.status.seqActive )
      wire#w1
      Coil( "Unit1.Em1.ControlNodes".unWinder."step".action[301] )
   END_RUNG
   RUNG wire#w1
      Coil( "Unit1.Em1.ControlNodes".unWinder."step".transition[301] )
   END_RUNG
   RUNG wire#w1
      Contact( "Unit1.Em1.ControlNodes".unWinder."step".transition[301] )
      { S7_Templates := "time_type := Time" } #statTonTimer[301].TON(pt := #SeqNoDelayTime, et =>)
      Move(in := #JOB_3_STEP_11, out1 => "Unit1.Em1.ControlNodes".unWinder.sequence.status.nextStep)
   END_RUNG
   // the same network as SCL:
   "Unit1.Em1.ControlNodes".unWinder."step".action[301] := ("Unit1.Em1.ControlNodes".unWinder.sequence.status.currentStep = #JOB_3_STEP_01) AND "Unit1.Em1.ControlNodes".unWinder.sequence.status.seqActive;
   "Unit1.Em1.ControlNodes".unWinder."step".transition[301] := ("Unit1.Em1.ControlNodes".unWinder.sequence.status.currentStep = #JOB_3_STEP_01) AND "Unit1.Em1.ControlNodes".unWinder.sequence.status.seqActive;
   #statTonTimer[301].TON(IN := ("Unit1.Em1.ControlNodes".unWinder.sequence.status.currentStep = #JOB_3_STEP_01) AND "Unit1.Em1.ControlNodes".unWinder.sequence.status.seqActive AND "Unit1.Em1.ControlNodes".unWinder."step".transition[301],
                          PT := #SeqNoDelayTime);
   IF #statTonTimer[301].Q THEN
       "Unit1.Em1.ControlNodes".unWinder.sequence.status.nextStep := #JOB_3_STEP_11;
   END_IF;
END_REGION

REGION Network 23: Step[311] : LConSMC_Winder speedMatch Command
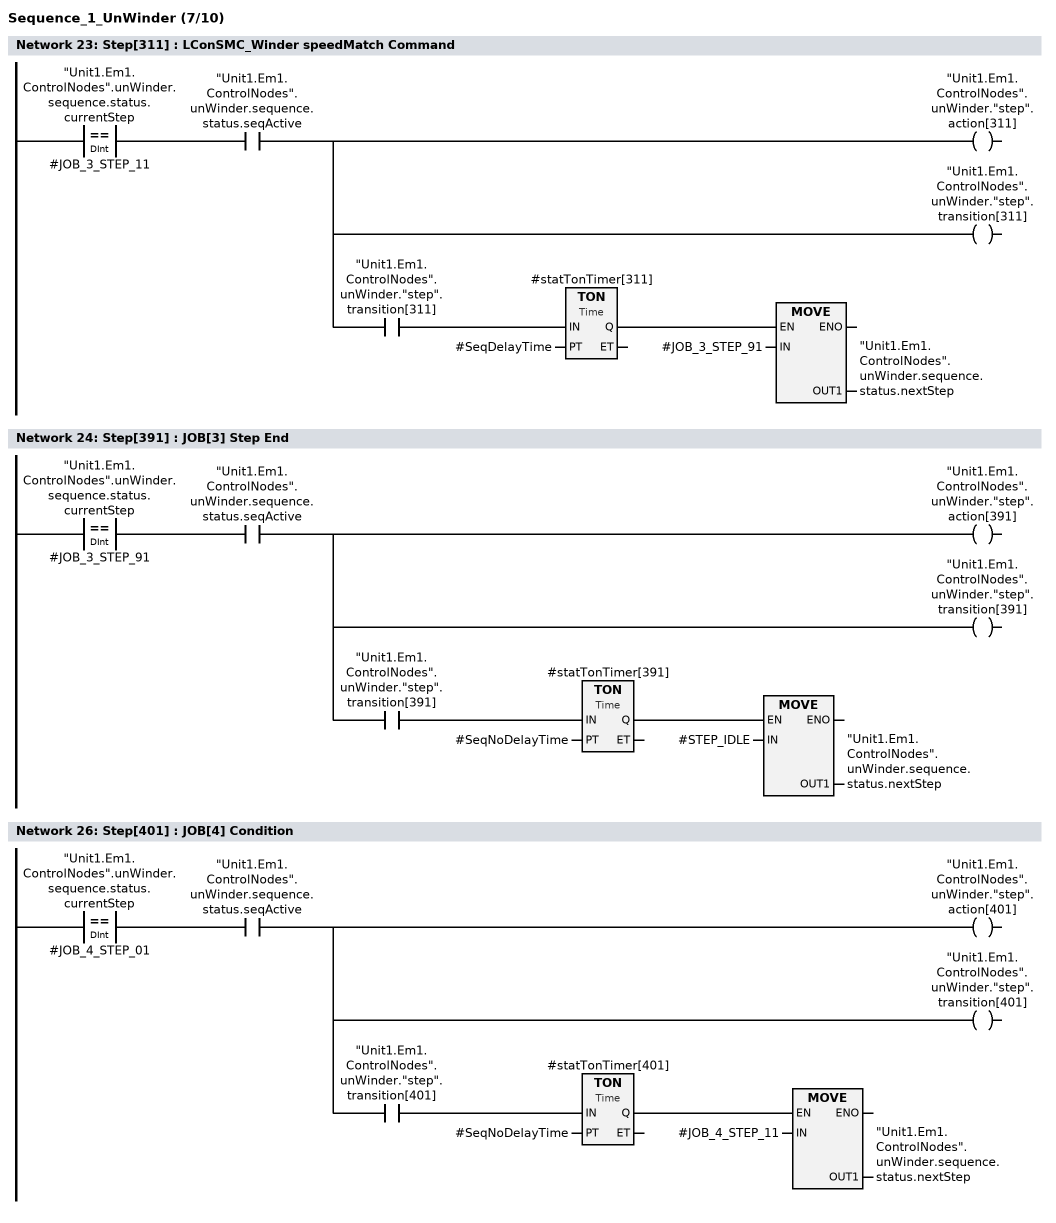
   RUNG wire#powerrail
      { S7_Templates := "SrcType := DInt" } EQ_Contact(in1 := "Unit1.Em1.ControlNodes".unWinder.sequence.status.currentStep, in2 := #JOB_3_STEP_11)
      Contact( "Unit1.Em1.ControlNodes".unWinder.sequence.status.seqActive )
      wire#w1
      Coil( "Unit1.Em1.ControlNodes".unWinder."step".action[311] )
   END_RUNG
   RUNG wire#w1
      Coil( "Unit1.Em1.ControlNodes".unWinder."step".transition[311] )
   END_RUNG
   RUNG wire#w1
      Contact( "Unit1.Em1.ControlNodes".unWinder."step".transition[311] )
      { S7_Templates := "time_type := Time" } #statTonTimer[311].TON(pt := #SeqDelayTime, et =>)
      Move(in := #JOB_3_STEP_91, out1 => "Unit1.Em1.ControlNodes".unWinder.sequence.status.nextStep)
   END_RUNG
   // the same network as SCL:
   "Unit1.Em1.ControlNodes".unWinder."step".action[311] := ("Unit1.Em1.ControlNodes".unWinder.sequence.status.currentStep = #JOB_3_STEP_11) AND "Unit1.Em1.ControlNodes".unWinder.sequence.status.seqActive;
   "Unit1.Em1.ControlNodes".unWinder."step".transition[311] := ("Unit1.Em1.ControlNodes".unWinder.sequence.status.currentStep = #JOB_3_STEP_11) AND "Unit1.Em1.ControlNodes".unWinder.sequence.status.seqActive;
   #statTonTimer[311].TON(IN := ("Unit1.Em1.ControlNodes".unWinder.sequence.status.currentStep = #JOB_3_STEP_11) AND "Unit1.Em1.ControlNodes".unWinder.sequence.status.seqActive AND "Unit1.Em1.ControlNodes".unWinder."step".transition[311],
                          PT := #SeqDelayTime);
   IF #statTonTimer[311].Q THEN
       "Unit1.Em1.ControlNodes".unWinder.sequence.status.nextStep := #JOB_3_STEP_91;
   END_IF;
END_REGION

REGION Network 24: Step[391] : JOB[3] Step End
   RUNG wire#powerrail
      { S7_Templates := "SrcType := DInt" } EQ_Contact(in1 := "Unit1.Em1.ControlNodes".unWinder.sequence.status.currentStep, in2 := #JOB_3_STEP_91)
      Contact( "Unit1.Em1.ControlNodes".unWinder.sequence.status.seqActive )
      wire#w1
      Coil( "Unit1.Em1.ControlNodes".unWinder."step".action[391] )
   END_RUNG
   RUNG wire#w1
      Coil( "Unit1.Em1.ControlNodes".unWinder."step".transition[391] )
   END_RUNG
   RUNG wire#w1
      Contact( "Unit1.Em1.ControlNodes".unWinder."step".transition[391] )
      { S7_Templates := "time_type := Time" } #statTonTimer[391].TON(pt := #SeqNoDelayTime, et =>)
      Move(in := #STEP_IDLE, out1 => "Unit1.Em1.ControlNodes".unWinder.sequence.status.nextStep)
   END_RUNG
   // the same network as SCL:
   "Unit1.Em1.ControlNodes".unWinder."step".action[391] := ("Unit1.Em1.ControlNodes".unWinder.sequence.status.currentStep = #JOB_3_STEP_91) AND "Unit1.Em1.ControlNodes".unWinder.sequence.status.seqActive;
   "Unit1.Em1.ControlNodes".unWinder."step".transition[391] := ("Unit1.Em1.ControlNodes".unWinder.sequence.status.currentStep = #JOB_3_STEP_91) AND "Unit1.Em1.ControlNodes".unWinder.sequence.status.seqActive;
   #statTonTimer[391].TON(IN := ("Unit1.Em1.ControlNodes".unWinder.sequence.status.currentStep = #JOB_3_STEP_91) AND "Unit1.Em1.ControlNodes".unWinder.sequence.status.seqActive AND "Unit1.Em1.ControlNodes".unWinder."step".transition[391],
                          PT := #SeqNoDelayTime);
   IF #statTonTimer[391].Q THEN
       "Unit1.Em1.ControlNodes".unWinder.sequence.status.nextStep := #STEP_IDLE;
   END_IF;
END_REGION

REGION Network 25: ******************** JOB[4] UNWINDER REWINDING ********************
END_REGION

REGION Network 26: Step[401] : JOB[4] Condition
   RUNG wire#powerrail
      { S7_Templates := "SrcType := DInt" } EQ_Contact(in1 := "Unit1.Em1.ControlNodes".unWinder.sequence.status.currentStep, in2 := #JOB_4_STEP_01)
      Contact( "Unit1.Em1.ControlNodes".unWinder.sequence.status.seqActive )
      wire#w1
      Coil( "Unit1.Em1.ControlNodes".unWinder."step".action[401] )
   END_RUNG
   RUNG wire#w1
      Coil( "Unit1.Em1.ControlNodes".unWinder."step".transition[401] )
   END_RUNG
   RUNG wire#w1
      Contact( "Unit1.Em1.ControlNodes".unWinder."step".transition[401] )
      { S7_Templates := "time_type := Time" } #statTonTimer[401].TON(pt := #SeqNoDelayTime, et =>)
      Move(in := #JOB_4_STEP_11, out1 => "Unit1.Em1.ControlNodes".unWinder.sequence.status.nextStep)
   END_RUNG
   // the same network as SCL:
   "Unit1.Em1.ControlNodes".unWinder."step".action[401] := ("Unit1.Em1.ControlNodes".unWinder.sequence.status.currentStep = #JOB_4_STEP_01) AND "Unit1.Em1.ControlNodes".unWinder.sequence.status.seqActive;
   "Unit1.Em1.ControlNodes".unWinder."step".transition[401] := ("Unit1.Em1.ControlNodes".unWinder.sequence.status.currentStep = #JOB_4_STEP_01) AND "Unit1.Em1.ControlNodes".unWinder.sequence.status.seqActive;
   #statTonTimer[401].TON(IN := ("Unit1.Em1.ControlNodes".unWinder.sequence.status.currentStep = #JOB_4_STEP_01) AND "Unit1.Em1.ControlNodes".unWinder.sequence.status.seqActive AND "Unit1.Em1.ControlNodes".unWinder."step".transition[401],
                          PT := #SeqNoDelayTime);
   IF #statTonTimer[401].Q THEN
       "Unit1.Em1.ControlNodes".unWinder.sequence.status.nextStep := #JOB_4_STEP_11;
   END_IF;
END_REGION

REGION Network 27: Step[411] : LConSMC_Winder Jog BackWard Command
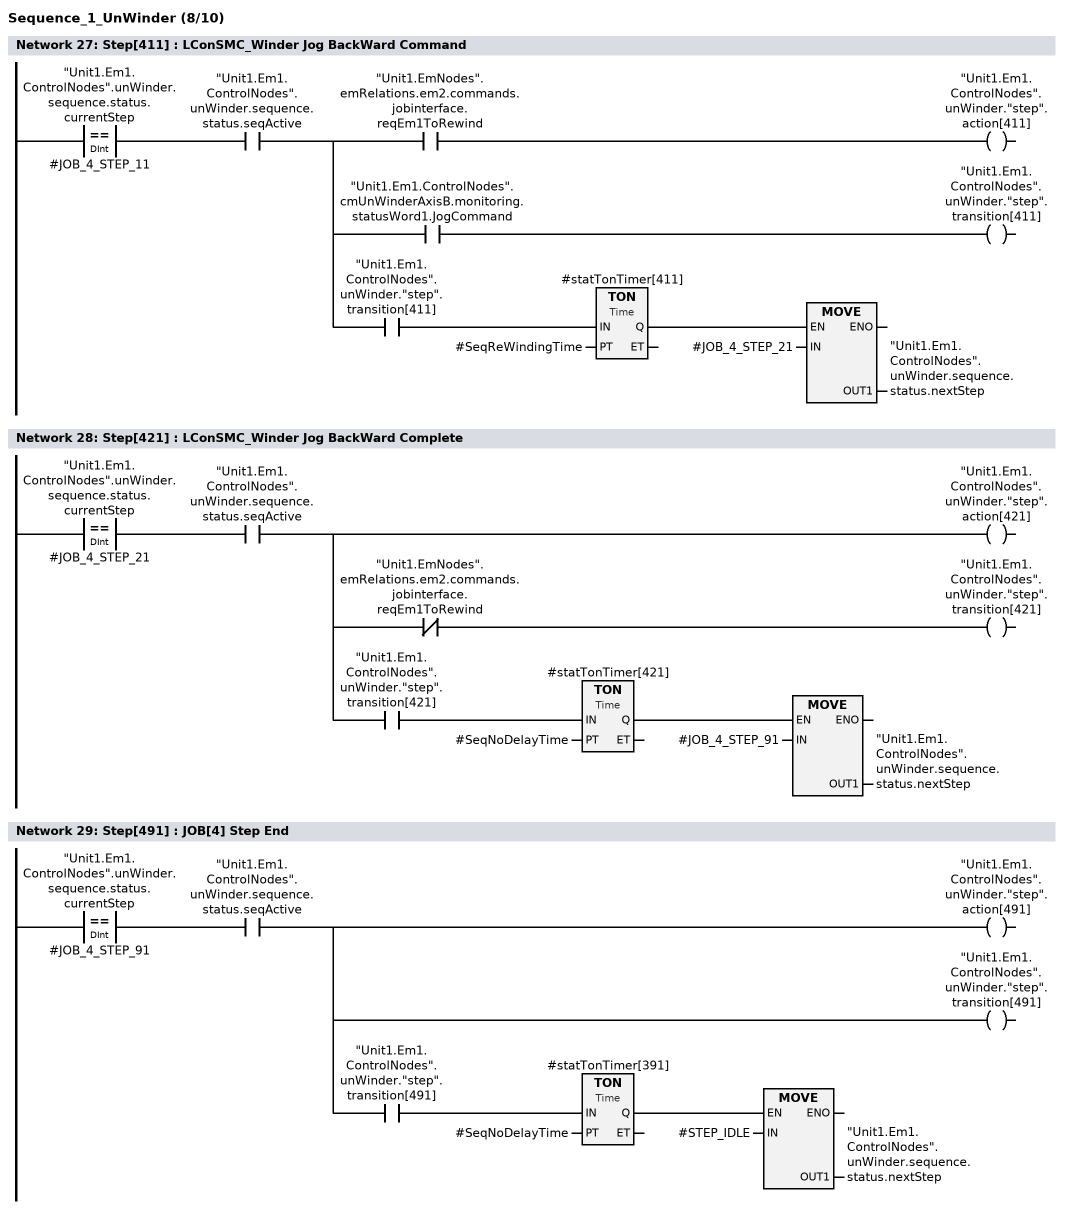
   RUNG wire#powerrail
      { S7_Templates := "SrcType := DInt" } EQ_Contact(in1 := "Unit1.Em1.ControlNodes".unWinder.sequence.status.currentStep, in2 := #JOB_4_STEP_11)
      Contact( "Unit1.Em1.ControlNodes".unWinder.sequence.status.seqActive )
      wire#w1
      Contact( "Unit1.EmNodes".emRelations.em2.commands.jobinterface.reqEm1ToRewind )
      Coil( "Unit1.Em1.ControlNodes".unWinder."step".action[411] )
   END_RUNG
   RUNG wire#w1
      Contact( "Unit1.Em1.ControlNodes".cmUnWinderAxisB.monitoring.statusWord1.JogCommand )
      Coil( "Unit1.Em1.ControlNodes".unWinder."step".transition[411] )
   END_RUNG
   RUNG wire#w1
      Contact( "Unit1.Em1.ControlNodes".unWinder."step".transition[411] )
      { S7_Templates := "time_type := Time" } #statTonTimer[411].TON(pt := #SeqReWindingTime, et =>)
      Move(in := #JOB_4_STEP_21, out1 => "Unit1.Em1.ControlNodes".unWinder.sequence.status.nextStep)
   END_RUNG
   // the same network as SCL:
   #_w1 := ("Unit1.Em1.ControlNodes".unWinder.sequence.status.currentStep = #JOB_4_STEP_11) AND "Unit1.Em1.ControlNodes".unWinder.sequence.status.seqActive;
   "Unit1.Em1.ControlNodes".unWinder."step".action[411] := #_w1 AND "Unit1.EmNodes".emRelations.em2.commands.jobinterface.reqEm1ToRewind;
   "Unit1.Em1.ControlNodes".unWinder."step".transition[411] := #_w1 AND "Unit1.Em1.ControlNodes".cmUnWinderAxisB.monitoring.statusWord1.JogCommand;
   #statTonTimer[411].TON(IN := #_w1 AND "Unit1.Em1.ControlNodes".unWinder."step".transition[411],
                          PT := #SeqReWindingTime);
   IF #statTonTimer[411].Q THEN
       "Unit1.Em1.ControlNodes".unWinder.sequence.status.nextStep := #JOB_4_STEP_21;
   END_IF;
END_REGION

REGION Network 28: Step[421] : LConSMC_Winder Jog BackWard Complete
   RUNG wire#powerrail
      { S7_Templates := "SrcType := DInt" } EQ_Contact(in1 := "Unit1.Em1.ControlNodes".unWinder.sequence.status.currentStep, in2 := #JOB_4_STEP_21)
      Contact( "Unit1.Em1.ControlNodes".unWinder.sequence.status.seqActive )
      wire#w1
      Coil( "Unit1.Em1.ControlNodes".unWinder."step".action[421] )
   END_RUNG
   RUNG wire#w1
      I_Contact( "Unit1.EmNodes".emRelations.em2.commands.jobinterface.reqEm1ToRewind )
      Coil( "Unit1.Em1.ControlNodes".unWinder."step".transition[421] )
   END_RUNG
   RUNG wire#w1
      Contact( "Unit1.Em1.ControlNodes".unWinder."step".transition[421] )
      { S7_Templates := "time_type := Time" } #statTonTimer[421].TON(pt := #SeqNoDelayTime, et =>)
      Move(in := #JOB_4_STEP_91, out1 => "Unit1.Em1.ControlNodes".unWinder.sequence.status.nextStep)
   END_RUNG
   // the same network as SCL:
   "Unit1.Em1.ControlNodes".unWinder."step".action[421] := ("Unit1.Em1.ControlNodes".unWinder.sequence.status.currentStep = #JOB_4_STEP_21) AND "Unit1.Em1.ControlNodes".unWinder.sequence.status.seqActive;
   "Unit1.Em1.ControlNodes".unWinder."step".transition[421] := ("Unit1.Em1.ControlNodes".unWinder.sequence.status.currentStep = #JOB_4_STEP_21) AND "Unit1.Em1.ControlNodes".unWinder.sequence.status.seqActive AND NOT "Unit1.EmNodes".emRelations.em2.commands.jobinterface.reqEm1ToRewind;
   #statTonTimer[421].TON(IN := ("Unit1.Em1.ControlNodes".unWinder.sequence.status.currentStep = #JOB_4_STEP_21) AND "Unit1.Em1.ControlNodes".unWinder.sequence.status.seqActive AND "Unit1.Em1.ControlNodes".unWinder."step".transition[421],
                          PT := #SeqNoDelayTime);
   IF #statTonTimer[421].Q THEN
       "Unit1.Em1.ControlNodes".unWinder.sequence.status.nextStep := #JOB_4_STEP_91;
   END_IF;
END_REGION

REGION Network 29: Step[491] : JOB[4] Step End
   RUNG wire#powerrail
      { S7_Templates := "SrcType := DInt" } EQ_Contact(in1 := "Unit1.Em1.ControlNodes".unWinder.sequence.status.currentStep, in2 := #JOB_4_STEP_91)
      Contact( "Unit1.Em1.ControlNodes".unWinder.sequence.status.seqActive )
      wire#w1
      Coil( "Unit1.Em1.ControlNodes".unWinder."step".action[491] )
   END_RUNG
   RUNG wire#w1
      Coil( "Unit1.Em1.ControlNodes".unWinder."step".transition[491] )
   END_RUNG
   RUNG wire#w1
      Contact( "Unit1.Em1.ControlNodes".unWinder."step".transition[491] )
      { S7_Templates := "time_type := Time" } #statTonTimer[391].TON(pt := #SeqNoDelayTime, et =>)
      Move(in := #STEP_IDLE, out1 => "Unit1.Em1.ControlNodes".unWinder.sequence.status.nextStep)
   END_RUNG
   // the same network as SCL:
   "Unit1.Em1.ControlNodes".unWinder."step".action[491] := ("Unit1.Em1.ControlNodes".unWinder.sequence.status.currentStep = #JOB_4_STEP_91) AND "Unit1.Em1.ControlNodes".unWinder.sequence.status.seqActive;
   "Unit1.Em1.ControlNodes".unWinder."step".transition[491] := ("Unit1.Em1.ControlNodes".unWinder.sequence.status.currentStep = #JOB_4_STEP_91) AND "Unit1.Em1.ControlNodes".unWinder.sequence.status.seqActive;
   #statTonTimer[391].TON(IN := ("Unit1.Em1.ControlNodes".unWinder.sequence.status.currentStep = #JOB_4_STEP_91) AND "Unit1.Em1.ControlNodes".unWinder.sequence.status.seqActive AND "Unit1.Em1.ControlNodes".unWinder."step".transition[491],
                          PT := #SeqNoDelayTime);
   IF #statTonTimer[391].Q THEN
       "Unit1.Em1.ControlNodes".unWinder.sequence.status.nextStep := #STEP_IDLE;
   END_IF;
END_REGION

REGION Network 30: ******************** IMMEDIATE STOP ********************
END_REGION

REGION Network 31: Immediate Stop
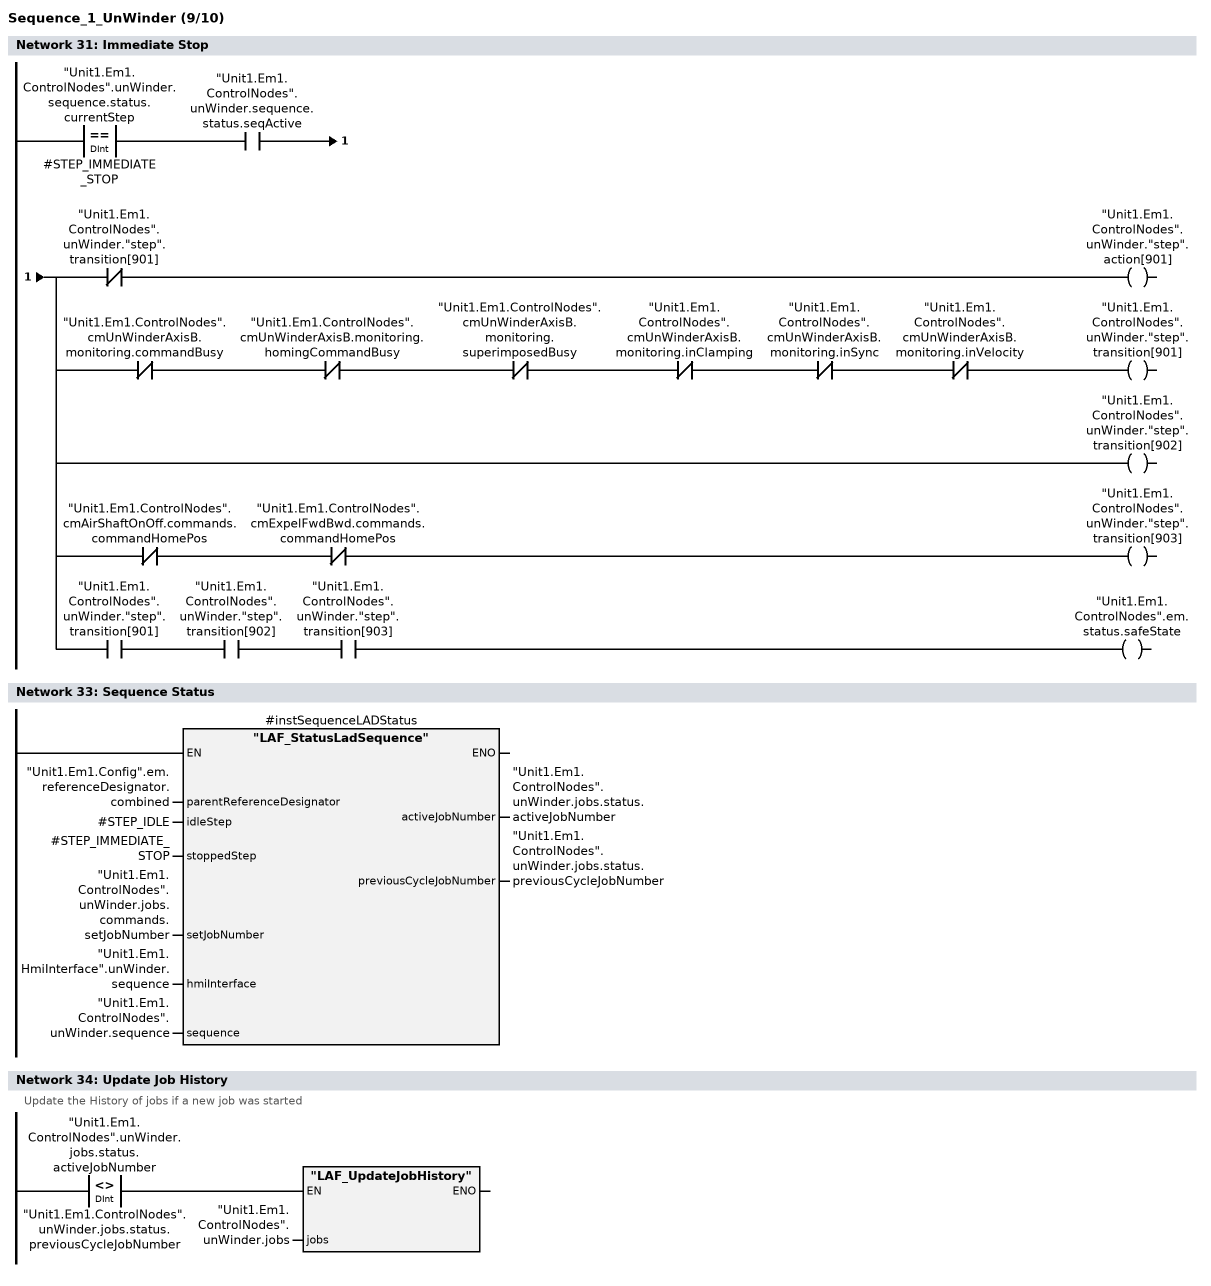
   RUNG wire#powerrail
      { S7_Templates := "SrcType := DInt" } EQ_Contact(in1 := "Unit1.Em1.ControlNodes".unWinder.sequence.status.currentStep, in2 := #STEP_IMMEDIATE_STOP)
      Contact( "Unit1.Em1.ControlNodes".unWinder.sequence.status.seqActive )
      wire#w1
      I_Contact( "Unit1.Em1.ControlNodes".unWinder."step".transition[901] )
      Coil( "Unit1.Em1.ControlNodes".unWinder."step".action[901] )
   END_RUNG
   RUNG wire#w1
      I_Contact( "Unit1.Em1.ControlNodes".cmUnWinderAxisB.monitoring.commandBusy )
      I_Contact( "Unit1.Em1.ControlNodes".cmUnWinderAxisB.monitoring.homingCommandBusy )
      I_Contact( "Unit1.Em1.ControlNodes".cmUnWinderAxisB.monitoring.superimposedBusy )
      I_Contact( "Unit1.Em1.ControlNodes".cmUnWinderAxisB.monitoring.inClamping )
      I_Contact( "Unit1.Em1.ControlNodes".cmUnWinderAxisB.monitoring.inSync )
      I_Contact( "Unit1.Em1.ControlNodes".cmUnWinderAxisB.monitoring.inVelocity )
      Coil( "Unit1.Em1.ControlNodes".unWinder."step".transition[901] )
   END_RUNG
   RUNG wire#w1
      Coil( "Unit1.Em1.ControlNodes".unWinder."step".transition[902] )
   END_RUNG
   RUNG wire#w1
      I_Contact( "Unit1.Em1.ControlNodes".cmAirShaftOnOff.commands.commandHomePos )
      I_Contact( "Unit1.Em1.ControlNodes".cmExpelFwdBwd.commands.commandHomePos )
      Coil( "Unit1.Em1.ControlNodes".unWinder."step".transition[903] )
   END_RUNG
   RUNG wire#w1
      Contact( "Unit1.Em1.ControlNodes".unWinder."step".transition[901] )
      Contact( "Unit1.Em1.ControlNodes".unWinder."step".transition[902] )
      Contact( "Unit1.Em1.ControlNodes".unWinder."step".transition[903] )
      Coil( "Unit1.Em1.ControlNodes".em.status.safeState )
   END_RUNG
   // the same network as SCL:
   #_w1 := ("Unit1.Em1.ControlNodes".unWinder.sequence.status.currentStep = #STEP_IMMEDIATE_STOP) AND "Unit1.Em1.ControlNodes".unWinder.sequence.status.seqActive;
   "Unit1.Em1.ControlNodes".unWinder."step".action[901] := #_w1 AND NOT "Unit1.Em1.ControlNodes".unWinder."step".transition[901];
   "Unit1.Em1.ControlNodes".unWinder."step".transition[901] := #_w1 AND NOT "Unit1.Em1.ControlNodes".cmUnWinderAxisB.monitoring.commandBusy AND NOT "Unit1.Em1.ControlNodes".cmUnWinderAxisB.monitoring.homingCommandBusy AND NOT "Unit1.Em1.ControlNodes".cmUnWinderAxisB.monitoring.superimposedBusy AND NOT "Unit1.Em1.ControlNodes".cmUnWinderAxisB.monitoring.inClamping AND NOT "Unit1.Em1.ControlNodes".cmUnWinderAxisB.monitoring.inSync AND NOT "Unit1.Em1.ControlNodes".cmUnWinderAxisB.monitoring.inVelocity;
   "Unit1.Em1.ControlNodes".unWinder."step".transition[902] := #_w1;
   "Unit1.Em1.ControlNodes".unWinder."step".transition[903] := #_w1 AND NOT "Unit1.Em1.ControlNodes".cmAirShaftOnOff.commands.commandHomePos AND NOT "Unit1.Em1.ControlNodes".cmExpelFwdBwd.commands.commandHomePos;
   "Unit1.Em1.ControlNodes".em.status.safeState := #_w1 AND "Unit1.Em1.ControlNodes".unWinder."step".transition[901] AND "Unit1.Em1.ControlNodes".unWinder."step".transition[902] AND "Unit1.Em1.ControlNodes".unWinder."step".transition[903];
END_REGION

REGION Network 32: ******************** STATUS ********************
END_REGION

REGION Network 33: Sequence Status
   RUNG wire#powerrail
      #instSequenceLADStatus(parentReferenceDesignator := "Unit1.Em1.Config".em.referenceDesignator.combined, idleStep := #STEP_IDLE, stoppedStep := #STEP_IMMEDIATE_STOP, setJobNumber := "Unit1.Em1.ControlNodes".unWinder.jobs.commands.setJobNumber, hmiInterface := "Unit1.Em1.HmiInterface".unWinder.sequence, sequence := "Unit1.Em1.ControlNodes".unWinder.sequence, activeJobNumber => "Unit1.Em1.ControlNodes".unWinder.jobs.status.activeJobNumber, previousCycleJobNumber => "Unit1.Em1.ControlNodes".unWinder.jobs.status.previousCycleJobNumber)
   END_RUNG
   // the same network as SCL:
   #instSequenceLADStatus(parentReferenceDesignator := "Unit1.Em1.Config".em.referenceDesignator.combined,   // "LAF_StatusLadSequence"
                          idleStep := #STEP_IDLE,
                          stoppedStep := #STEP_IMMEDIATE_STOP,
                          setJobNumber := "Unit1.Em1.ControlNodes".unWinder.jobs.commands.setJobNumber,
                          hmiInterface := "Unit1.Em1.HmiInterface".unWinder.sequence,
                          sequence := "Unit1.Em1.ControlNodes".unWinder.sequence,
                          activeJobNumber => "Unit1.Em1.ControlNodes".unWinder.jobs.status.activeJobNumber,
                          previousCycleJobNumber => "Unit1.Em1.ControlNodes".unWinder.jobs.status.previousCycleJobNumber);
END_REGION

REGION Network 34: Update Job History
   // Update the History of jobs if a new job was started
   RUNG wire#powerrail
      { S7_Templates := "SrcType := DInt" } NE_Contact(in1 := "Unit1.Em1.ControlNodes".unWinder.jobs.status.activeJobNumber, in2 := "Unit1.Em1.ControlNodes".unWinder.jobs.status.previousCycleJobNumber)
      "LAF_UpdateJobHistory"(jobs := "Unit1.Em1.ControlNodes".unWinder.jobs)
   END_RUNG
   // the same network as SCL:
   IF "Unit1.Em1.ControlNodes".unWinder.jobs.status.activeJobNumber <> "Unit1.Em1.ControlNodes".unWinder.jobs.status.previousCycleJobNumber THEN
       "LAF_UpdateJobHistory"(jobs := "Unit1.Em1.ControlNodes".unWinder.jobs);
   END_IF;
END_REGION

REGION Network 35: Output steps as String
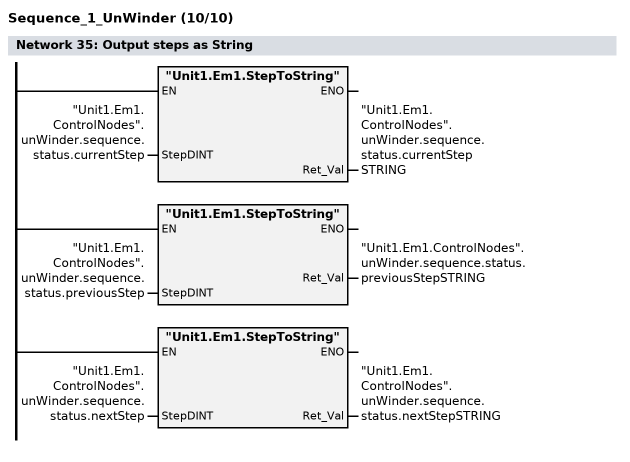
   RUNG wire#powerrail
      "Unit1.Em1.StepToString"(StepDINT := "Unit1.Em1.ControlNodes".unWinder.sequence.status.currentStep, Ret_Val => "Unit1.Em1.ControlNodes".unWinder.sequence.status.currentStepSTRING)
   END_RUNG
   RUNG wire#powerrail
      "Unit1.Em1.StepToString"(StepDINT := "Unit1.Em1.ControlNodes".unWinder.sequence.status.previousStep, Ret_Val => "Unit1.Em1.ControlNodes".unWinder.sequence.status.previousStepSTRING)
   END_RUNG
   RUNG wire#powerrail
      "Unit1.Em1.StepToString"(StepDINT := "Unit1.Em1.ControlNodes".unWinder.sequence.status.nextStep, Ret_Val => "Unit1.Em1.ControlNodes".unWinder.sequence.status.nextStepSTRING)
   END_RUNG
   // the same network as SCL:
   "Unit1.Em1.ControlNodes".unWinder.sequence.status.currentStepSTRING := "Unit1.Em1.StepToString"(StepDINT := "Unit1.Em1.ControlNodes".unWinder.sequence.status.currentStep);
   "Unit1.Em1.ControlNodes".unWinder.sequence.status.previousStepSTRING := "Unit1.Em1.StepToString"(StepDINT := "Unit1.Em1.ControlNodes".unWinder.sequence.status.previousStep);
   "Unit1.Em1.ControlNodes".unWinder.sequence.status.nextStepSTRING := "Unit1.Em1.StepToString"(StepDINT := "Unit1.Em1.ControlNodes".unWinder.sequence.status.nextStep);
END_REGION
END_FUNCTION_BLOCK
